FUNCTION Convert_SINT_TO_TOD : BOOL
VAR_INPUT
	in : SINT;
	out : REFERENCE TO TOD;
END_VAR
VAR
	converted : TOD;
END_VAR

converted := SINT_TO_TOD(in);

IF (TOD_TO_SINT(converted) <> in) THEN
	RETURN;
END_IF

out := converted;
Convert_SINT_TO_TOD := TRUE;

END_FUNCTION

(* stored: Version 1.1.0.1, ProductVersion 3.1.4024.12
   POU Convert_SINT_TO_TOD: Id {005be8a2-7f3b-4433-9fb0-4a2e38b878c5}, SpecialFunc None *)
